# EPICS autosave request: motorApp/Db/positionCompare_settings.req
$(P)$(R)PCOStartPosition
$(P)$(R)PCOEndPosition
$(P)$(R)PCOIncrement
$(P)$(R)PCOPulseWidth
